PROGRAM PRG_Compilation
VAR
END_VAR

END_PROGRAM

(* stored: Version 1.1.0.1
   POU PRG_Compilation: Id {e3d1aff8-90e2-4b06-bf62-3f7b8a8c4d92}, SpecialFunc None *)
